# EPICS autosave request: iocBoot/gmca_23i_ioc1/dbSave/BP_Kb_.req
%
% BURT Request File
%
% $(P)BP:Kb:  BPM @ KB mirrors position
%
file assy.req ASSY=$(P)BP:Kb
file mtr1.req MTR1=$(P)BP:mkb
file drv1.req DRV1=$(P)BP:KBZ

$(P)BP:KBZ:RqsPosMem1
$(P)BP:KBZ:RqsPosMem2
$(P)BP:KBZ:RqsPosMem3

$(P)BP:KBZ:RqsPosMem1.DESC
$(P)BP:KBZ:RqsPosMem2.DESC
$(P)BP:KBZ:RqsPosMem3.DESC
